FUNCTION_BLOCK AppContext EXTENDS TcoCore.TcoContext
VAR
    _mainStation : MainStation(THIS^);

    {attribute addProperty Name "Versionsnummer Plc"}
    _sVersion : STRING(23);
    //~
    _stProgramVersion : ST_LibVersion;
    //~

END_VAR

(*~
    <docu>
        <summary>
            Main method of the TcoContext. This is the entry point of any control logic that belongs to this context.
            The call of this method is ensured by calling the <c>InstanceName.Run()</c> method, and it must not be called explicitly.
            This method is abstract, and it must be overridden in derived block.
        </summary>
    </docu>
~*)
METHOD PROTECTED Main
_mainStation();

//IF (THIS^._startCycleCount MOD 10 = 0) THEN
//    Logger.Push('This is a log entry', eMessageCategory.Trace);
//END_IF;

//IF (THIS^._startCycleCount MOD 125 = 0) THEN
//    Logger.Push('This is a log entry', eMessageCategory.Info);
//END_IF;

//IF (THIS^._startCycleCount MOD 400 = 0) THEN
//    Logger.Push('This is a log entry', eMessageCategory.Warning);
//END_IF;

//IF (THIS^._startCycleCount MOD 2000 = 0) THEN
//    Logger.Push('This is a log entry', eMessageCategory.Error);
//END_IF;
END_METHOD

END_FUNCTION_BLOCK

(* stored: Version 1.1.0.1, ProductVersion 3.1.4024.12
   POU AppContext: Id {39f0217b-7a4b-0a4f-0c8f-c7e3dcadd944}, SpecialFunc None
   Method Main: Id {caf3358f-a01c-0f58-099c-46db5a23cb11} *)
